Staubli VAL3: fbkStreamer.pgx

public program fbkStreamer()
begin
  //bStream = true
  call setupRosMsgs()
  //while (bStream)
  while (true)
    // fetch robot status
    //call fetchStatus()

    // encode and send ROS simple message ID 13: robot status
    //call encodeStatus()
    //call sendRosMsg(rosMsgStatus)

    // fetch current joint values
    jCurrPose=herej()

    // encode and send ROS simple_message ID 15: joint feedback
    call encodeJointFbk()
    call sendJointFbk()
    delay(0)
  endWhile
end
